// TIA Portal V17 export
// export: Created 2024-06-16T17:47:25.0978867Z, ExportSetting WithDefaults, DisplayName Totally Integrated Automation Portal, DisplayVersion V17, DisplayName TIA Portal Openness, DisplayVersion V17, DisplayName TIA Portal Version Control Interface, DisplayVersion V17, DisplayName STEP 7 Professional, DisplayVersion V17, DisplayName STEP 7 Safety, DisplayVersion V17, DisplayName WinCC Professional, DisplayVersion V17
DATA_BLOCK "St1_Out"   // DB115
{ S7_Optimized_Access := 'TRUE' }
VERSION : 0.1
// stored: AutoNumber false, DBAccessibleFromOPCUA true, DBAccessibleFromWebserver true, IsOnlyStoredInLoadMemory false, IsRetainMemResEnabled false, IsWriteProtectedInAS false, MemoryReserve 100
   VAR
      Ouverture_Pinces : Bool;   // Ouverture : Pinces de préhension
      Fermeture_Pinces : Bool;   // Fermeture : Pinces de préhension
      Vy_PileAV : Bool;   // Conditions sur voyant C2 : OK
      Vy_PileAR : Bool;   // Conditions sur voyant C4 : OK
   END_VAR
BEGIN
END_DATA_BLOCK
